Yaskawa INFORM job: Souvenir barrenado.JBI

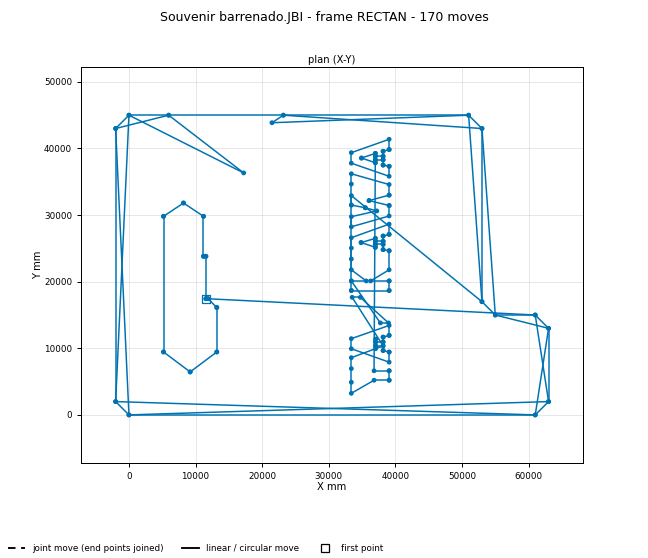
[picture p0: tool path of Souvenir barrenado.JBI in frame RECTAN, 170 of 170 moves have a stored position in this frame; points joined in program order, loops and branches not executed]
/JOB
//NAME SOUVENIR
//POS
///NPOS 7,0,0,0,0,0
///TOOL 0
///POSTYPE RECTAN
///RECTAN
C00000=11552,17453,0,0,0,0
C00001=11552,23816,0,0,0,0
C00002=11552,23816,0,0,0,0
C00003=11190,23816,0,0,0,0
C00004=11190,23816,0,0,0,0
C00005=11190,29816,0,0,0,0
C00006=11190,29816,0,0,0,0
C00007=8190,31816,0,0,0,0
C00008=8190,31816,0,0,0,0
C00009=5190,29816,0,0,0,0
C00010=5190,29816,0,0,0,0
C00011=5190,9453,0,0,0,0
C00012=5190,9453,0,0,0,0
C00013=9190,6453,0,0,0,0
C00014=9190,6453,0,0,0,0
C00015=13190,9453,0,0,0,0
C00016=13190,9453,0,0,0,0
C00017=13190,16125,0,0,0,0
C00018=13190,16125,0,0,0,0
C00019=11861,17453,0,0,0,0
C00020=11861,17453,0,0,0,0
C00021=11552,17453,0,0,0,0
C00022=61000,15000,0,0,0,0
C00023=55000,15000,0,0,0,0
C00024=63000,13000,0,0,0,0
C00025=61000,15000,0,0,0,0
C00026=63000,2000,0,0,0,0
C00027=63000,13000,0,0,0,0
C00028=61000,0,0,0,0,0
C00029=63000,2000,0,0,0,0
C00030=0,0,0,0,0,0
C00031=61000,0,0,0,0,0
C00032=-2000,2000,0,0,0,0
C00033=0,0,0,0,0,0
C00034=-2000,43000,0,0,0,0
C00035=-2000,2000,0,0,0,0
C00036=0,45000,0,0,0,0
C00037=-2000,43000,0,0,0,0
C00038=5963,45000,0,0,0,0
C00039=0,45000,0,0,0,0
C00040=17225,36331,0,0,0,0
C00041=5963,45000,0,0,0,0
C00042=23182,45000,0,0,0,0
C00043=21469,43867,0,0,0,0
C00044=51000,45000,0,0,0,0
C00045=23182,45000,0,0,0,0
C00046=53000,43000,0,0,0,0
C00047=51000,45000,0,0,0,0
C00048=53000,17000,0,0,0,0
C00049=53000,43000,0,0,0,0
C00050=55000,15000,0,0,0,0
C00051=53000,17000,0,0,0,0
C00052=33386,32925,0,0,0,0
C00053=33386,31508,0,0,0,0
C00054=33386,31508,0,0,0,0
C00055=35485,31101,0,0,0,0
C00056=35485,31101,0,0,0,0
C00057=37217,30628,0,0,0,0
C00058=33386,29762,0,0,0,0
C00059=33386,28240,0,0,0,0
C00060=39063,29868,0,0,0,0
C00061=39063,31436,0,0,0,0
C00062=39063,31436,0,0,0,0
C00063=36053,32179,0,0,0,0
C00064=36053,32179,0,0,0,0
C00065=39063,32999,0,0,0,0
C00066=39063,32999,0,0,0,0
C00067=39063,34589,0,0,0,0
C00068=33386,36205,0,0,0,0
C00069=33386,34670,0,0,0,0
C00070=33386,20114,0,0,0,0
C00071=33386,18676,0,0,0,0
C00072=33386,18676,0,0,0,0
C00073=39063,18676,0,0,0,0
C00074=39063,18676,0,0,0,0
C00075=39063,20114,0,0,0,0
C00076=39063,20114,0,0,0,0
C00077=36282,20114,0,0,0,0
C00078=39063,21787,0,0,0,0
C00079=39063,24650,0,0,0,0
C00080=39063,24650,0,0,0,0
C00081=38159,24811,0,0,0,0
C00082=38159,24811,0,0,0,0
C00083=38159,25602,0,0,0,0
C00084=38159,25602,0,0,0,0
C00085=36991,25602,0,0,0,0
C00086=36991,25602,0,0,0,0
C00087=36991,25164,0,0,0,0
C00088=36991,25164,0,0,0,0
C00089=34855,25879,0,0,0,0
C00090=34855,25879,0,0,0,0
C00091=36991,26502,0,0,0,0
C00092=36991,26502,0,0,0,0
C00093=36991,26064,0,0,0,0
C00094=36991,26064,0,0,0,0
C00095=38159,26064,0,0,0,0
C00096=38159,26064,0,0,0,0
C00097=38159,26853,0,0,0,0
C00098=38159,26853,0,0,0,0
C00099=39063,27106,0,0,0,0
C00100=39063,27106,0,0,0,0
C00101=39063,28643,0,0,0,0
C00102=33386,26605,0,0,0,0
C00103=33386,25054,0,0,0,0
C00104=33386,23411,0,0,0,0
C00105=33386,21787,0,0,0,0
C00106=35625,20114,0,0,0,0
C00107=33386,20114,0,0,0,0
C00108=37739,13813,0,0,0,0
C00109=38965,13813,0,0,0,0
C00110=34736,17651,0,0,0,0
C00111=33511,17651,0,0,0,0
C00112=38159,10368,0,0,0,0
C00113=37033,10368,0,0,0,0
C00114=37033,10368,0,0,0,0
C00115=37033,9937,0,0,0,0
C00116=37033,11389,0,0,0,0
C00117=37033,10950,0,0,0,0
C00118=37033,10950,0,0,0,0
C00119=38159,10950,0,0,0,0
C00120=38159,10950,0,0,0,0
C00121=38159,11680,0,0,0,0
C00122=38159,11680,0,0,0,0
C00123=39063,11942,0,0,0,0
C00124=39063,11942,0,0,0,0
C00125=39063,13433,0,0,0,0
C00126=33386,11450,0,0,0,0
C00127=33386,9937,0,0,0,0
C00128=39063,7919,0,0,0,0
C00129=39063,9435,0,0,0,0
C00130=39063,9435,0,0,0,0
C00131=38159,9666,0,0,0,0
C00132=38159,9666,0,0,0,0
C00133=38159,10368,0,0,0,0
C00134=33386,8593,0,0,0,0
C00135=33386,6952,0,0,0,0
C00136=33386,4905,0,0,0,0
C00137=33386,3242,0,0,0,0
C00138=36797,5207,0,0,0,0
C00139=39063,5207,0,0,0,0
C00140=39063,5207,0,0,0,0
C00141=39063,6626,0,0,0,0
C00142=39063,6626,0,0,0,0
C00143=36797,6626,0,0,0,0
C00144=36991,38833,0,0,0,0
C00145=38159,38833,0,0,0,0
C00146=38159,38833,0,0,0,0
C00147=38159,39581,0,0,0,0
C00148=38159,39581,0,0,0,0
C00149=39063,39842,0,0,0,0
C00150=39063,39842,0,0,0,0
C00151=39063,41382,0,0,0,0
C00152=33386,39375,0,0,0,0
C00153=33386,37791,0,0,0,0
C00154=39063,35829,0,0,0,0
C00155=39063,37323,0,0,0,0
C00156=39063,37323,0,0,0,0
C00157=38159,37509,0,0,0,0
C00158=38159,37509,0,0,0,0
C00159=38159,38298,0,0,0,0
C00160=38159,38298,0,0,0,0
C00161=36991,38298,0,0,0,0
C00162=36991,38298,0,0,0,0
C00163=36991,37859,0,0,0,0
C00164=36991,37859,0,0,0,0
C00165=34914,38565,0,0,0,0
C00166=34914,38565,0,0,0,0
C00167=36991,39271,0,0,0,0
C00168=36991,39271,0,0,0,0
C00169=36991,38833,0,0,0,0
//INST
///DATE 2025/03/24 09:03
///ATTR SC,RW
///GROUP1 RB1
NOP
MOVJ C00000 VJ=25.00
MOVL C00001 V=83.3
MOVL C00002 V=83.3
MOVL C00003 V=83.3
MOVL C00004 V=83.3
MOVL C00005 V=83.3
MOVL C00006 V=83.3
MOVL C00007 V=83.3
MOVL C00008 V=83.3
MOVL C00009 V=83.3
MOVL C00010 V=83.3
MOVL C00011 V=83.3
MOVL C00012 V=83.3
MOVL C00013 V=83.3
MOVL C00014 V=83.3
MOVL C00015 V=83.3
MOVL C00016 V=83.3
MOVL C00017 V=83.3
MOVL C00018 V=83.3
MOVL C00019 V=83.3
MOVL C00020 V=83.3
MOVL C00021 V=83.3
MOVL C00022 V=83.3
MOVL C00023 V=83.3
MOVL C00024 V=83.3
MOVL C00025 V=83.3
MOVL C00026 V=83.3
MOVL C00027 V=83.3
MOVL C00028 V=83.3
MOVL C00029 V=83.3
MOVL C00030 V=83.3
MOVL C00031 V=83.3
MOVL C00032 V=83.3
MOVL C00033 V=83.3
MOVL C00034 V=83.3
MOVL C00035 V=83.3
MOVL C00036 V=83.3
MOVL C00037 V=83.3
MOVL C00038 V=83.3
MOVL C00039 V=83.3
MOVL C00040 V=83.3
MOVL C00041 V=83.3
MOVL C00042 V=83.3
MOVL C00043 V=83.3
MOVL C00044 V=83.3
MOVL C00045 V=83.3
MOVL C00046 V=83.3
MOVL C00047 V=83.3
MOVL C00048 V=83.3
MOVL C00049 V=83.3
MOVL C00050 V=83.3
MOVL C00051 V=83.3
MOVL C00052 V=83.3
MOVL C00053 V=83.3
MOVL C00054 V=83.3
MOVL C00055 V=83.3
MOVL C00056 V=83.3
MOVL C00057 V=83.3
MOVL C00058 V=83.3
MOVL C00059 V=83.3
MOVL C00060 V=83.3
MOVL C00061 V=83.3
MOVL C00062 V=83.3
MOVL C00063 V=83.3
MOVL C00064 V=83.3
MOVL C00065 V=83.3
MOVL C00066 V=83.3
MOVL C00067 V=83.3
MOVL C00068 V=83.3
MOVL C00069 V=83.3
MOVL C00070 V=83.3
MOVL C00071 V=83.3
MOVL C00072 V=83.3
MOVL C00073 V=83.3
MOVL C00074 V=83.3
MOVL C00075 V=83.3
MOVL C00076 V=83.3
MOVL C00077 V=83.3
MOVL C00078 V=83.3
MOVL C00079 V=83.3
MOVL C00080 V=83.3
MOVL C00081 V=83.3
MOVL C00082 V=83.3
MOVL C00083 V=83.3
MOVL C00084 V=83.3
MOVL C00085 V=83.3
MOVL C00086 V=83.3
MOVL C00087 V=83.3
MOVL C00088 V=83.3
MOVL C00089 V=83.3
MOVL C00090 V=83.3
MOVL C00091 V=83.3
MOVL C00092 V=83.3
MOVL C00093 V=83.3
MOVL C00094 V=83.3
MOVL C00095 V=83.3
MOVL C00096 V=83.3
MOVL C00097 V=83.3
MOVL C00098 V=83.3
MOVL C00099 V=83.3
MOVL C00100 V=83.3
MOVL C00101 V=83.3
MOVL C00102 V=83.3
MOVL C00103 V=83.3
MOVL C00104 V=83.3
MOVL C00105 V=83.3
MOVL C00106 V=83.3
MOVL C00107 V=83.3
MOVL C00108 V=83.3
MOVL C00109 V=83.3
MOVL C00110 V=83.3
MOVL C00111 V=83.3
MOVL C00112 V=83.3
MOVL C00113 V=83.3
MOVL C00114 V=83.3
MOVL C00115 V=83.3
MOVL C00116 V=83.3
MOVL C00117 V=83.3
MOVL C00118 V=83.3
MOVL C00119 V=83.3
MOVL C00120 V=83.3
MOVL C00121 V=83.3
MOVL C00122 V=83.3
MOVL C00123 V=83.3
MOVL C00124 V=83.3
MOVL C00125 V=83.3
MOVL C00126 V=83.3
MOVL C00127 V=83.3
MOVL C00128 V=83.3
MOVL C00129 V=83.3
MOVL C00130 V=83.3
MOVL C00131 V=83.3
MOVL C00132 V=83.3
MOVL C00133 V=83.3
MOVL C00134 V=83.3
MOVL C00135 V=83.3
MOVL C00136 V=83.3
MOVL C00137 V=83.3
MOVL C00138 V=83.3
MOVL C00139 V=83.3
MOVL C00140 V=83.3
MOVL C00141 V=83.3
MOVL C00142 V=83.3
MOVL C00143 V=83.3
MOVL C00144 V=83.3
MOVL C00145 V=83.3
MOVL C00146 V=83.3
MOVL C00147 V=83.3
MOVL C00148 V=83.3
MOVL C00149 V=83.3
MOVL C00150 V=83.3
MOVL C00151 V=83.3
MOVL C00152 V=83.3
MOVL C00153 V=83.3
MOVL C00154 V=83.3
MOVL C00155 V=83.3
MOVL C00156 V=83.3
MOVL C00157 V=83.3
MOVL C00158 V=83.3
MOVL C00159 V=83.3
MOVL C00160 V=83.3
MOVL C00161 V=83.3
MOVL C00162 V=83.3
MOVL C00163 V=83.3
MOVL C00164 V=83.3
MOVL C00165 V=83.3
MOVL C00166 V=83.3
MOVL C00167 V=83.3
MOVL C00168 V=83.3
MOVJ C00169 VJ=25.00
END
